PROGRAM PRG_ReadJsonFile
VAR
	eStateRead        : (R_STATE_IDLE, R_STATE_GET_SIZE, R_STATE_OPEN, R_STATE_READ, R_STATE_CLOSE, R_STATE_DONE, R_STATE_ERROR);
	nTotalBytesRead	  : UDINT;
	fbFileOpen        : FB_FileOpen;
	sFilePath         : T_MaxString;
	fbFormat   		  : FB_FormatString;
	udiFileHandle     : UINT;
	fbFileRead        : FB_FileRead;
	abReadBuffer      : ARRAY[0..1023] OF BYTE; (* Buffer para a leitura *)
	nBytesRead        : UDINT;
	fbFileClose       : FB_FileClose;
END_VAR

fbFormat(sFormat := 'C:\ProgramData\Beckhoff\TF2000 TwinCAT 3 HMI Server\service\TcHmiProject\www\DATA\Reports\%s', arg1:= F_STRING(in:= GVL_Report.testPath), sOut => sFilePath);

CASE eStateRead OF
    R_STATE_IDLE:
        IF GVL_Report.bStartRead THEN
            GVL_Report.bStartRead := FALSE;
            GVL_Report.sJsonOutput[0] := 0; (* Limpa a string de conteúdo antes de iniciar *)
			
			nTotalBytesRead	:= 0;
            eStateRead := R_STATE_OPEN;
        END_IF


    R_STATE_OPEN:
        fbFileOpen(
            bExecute    := TRUE,
            sNetId      := '',
            sPathName   := sFilePath,
            nMode       := FOPEN_MODEREAD, (* Modo de leitura de texto *)
            tTimeout    := T#5S);
            
        IF NOT fbFileOpen.bBusy THEN
            IF fbFileOpen.bError THEN
                eStateRead := R_STATE_ERROR;
            ELSE
                udiFileHandle := fbFileOpen.hFile;
                eStateRead := R_STATE_READ;
            END_IF
            fbFileOpen(bExecute := FALSE);
        END_IF

    R_STATE_READ:
       
		fbFileRead(
            bExecute    := TRUE,
            sNetId      := '',
            hFile 		:= udiFileHandle,
            pReadBuff   := ADR(abReadBuffer), (* Endereço do buffer temporário *)
            cbReadLen   := SIZEOF(abReadBuffer), (* Tamanho do buffer *)
            tTimeout    := T#5S);

        IF NOT fbFileRead.bBusy THEN
            IF fbFileRead.bError THEN
                eStateRead := R_STATE_ERROR;
            ELSE
                nBytesRead := fbFileRead.cbRead;
                IF nBytesRead > 0 THEN
                    (* Concatena a parte lida à string principal *)
                    MEMCPY(ADR(GVL_Report.sJsonOutput) + nTotalBytesRead, ADR(abReadBuffer), nBytesRead);
                    nTotalBytesRead := nTotalBytesRead + nBytesRead;
					
                    IF nBytesRead < SIZEOF(abReadBuffer) THEN
                        (* Fim do arquivo detectado (leu menos que o tamanho do buffer) *)
						GVL_Report.sJsonOutput[nTotalBytesRead] := 0;
                        eStateRead := R_STATE_CLOSE;
                    ELSE
                        (* Lê o próximo bloco no próximo ciclo *)
                        fbFileRead(bExecute := FALSE);
                    END_IF
                ELSE
                    (* nBytesRead é 0: Fim do arquivo *)
                    eStateRead := R_STATE_CLOSE;
                END_IF
            END_IF
        END_IF

    R_STATE_CLOSE:
        fbFileClose(
            bExecute    := TRUE,
            sNetId      := '',
            hFile 		:= udiFileHandle,
            tTimeout    := T#5S);
            
        IF NOT fbFileClose.bBusy THEN
            IF fbFileClose.bError THEN
                eStateRead := R_STATE_ERROR;
            ELSE
                eStateRead := R_STATE_DONE;
            END_IF
            fbFileClose(bExecute := FALSE);
        END_IF

    R_STATE_DONE:
        (* Leitura concluída. O conteúdo JSON está na variável sJsonContent. *)
        eStateRead := R_STATE_IDLE;
		GVL_Report.bGeneratePDF2:= TRUE;
		fbFileRead(bExecute := FALSE);

    R_STATE_ERROR:
        (* Tratar erro aqui. A variável fbFileGets.nErrId contém o código. *)
        eStateRead := R_STATE_IDLE;
END_CASE

END_PROGRAM

(* stored: Version 1.1.0.1, ProductVersion 3.1.4024.12
   POU PRG_ReadJsonFile: Id {c6628658-3b5f-4d45-81fe-0a3126adeb1e}, SpecialFunc None *)
